ABB RobotStudio station: welding.rspag

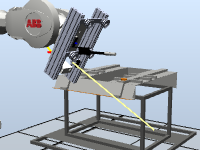
--- station ---
Station Solution21 (saved by RobotStudio format 3)
Controller IRB_7600_340kg_2.80m
  mechanical unit ROB_1: IRB7600_340_280__01, 6 joints, base frame (0, 0, 0) mm
Layout (positions relative to the parent item):
  - IRB7600_340_280__01 [mechanism, from Robots\IRB7600_340_280_G_01.rslib] at (0, 0, 0) mm; joint values [0, 0, 0, 0, 0.5236, 0] (rad or m)
  - Car Underbody [part]
  - Welding Gun [graphiccomponentgroup, from Libraries\Welding Gun.rslib] at (1932.51, 0, 1895) mm, rotated rx 180 ry 60 rz 180 deg
    - Part_1 [part, from Libraries\Welding Gun.rslib]
    - Part_2 [part, from Libraries\Welding Gun.rslib] at (-42.64, -13.71, 48.01) mm
    - Part_3 [part, from Libraries\Welding Gun.rslib] at (-42.16, -13.66, 198.7) mm, rotated rx 0 ry 60 rz 0 deg
    - Part_4 [part, from Libraries\Welding Gun.rslib] at (40.8, 0, 127.95) mm, rotated rx 0 ry -30 rz 0 deg
    - Part_6 [part, from Libraries\Welding Gun.rslib] at (-34.66, -7.16, 195.53) mm, rotated rx 0 ry 60 rz 0 deg
    - Part_8 [part, from Libraries\Welding Gun.rslib] at (-8.62, 0, 212.77) mm, rotated rx 0 ry -30 rz 0 deg
    - Part_9 [part, from Libraries\Welding Gun.rslib] at (-87.9, 0, 349.25) mm, rotated rx 0 ry -30 rz 0 deg
    - Part_10 [part, from Libraries\Welding Gun.rslib] at (-111.22, 0, 389.49) mm, rotated rx 0 ry -30 rz 0 deg
    - Part_11 [part, from Libraries\Welding Gun.rslib] at (-118.48, 0, 400.42) mm, rotated rx 0 ry -30 rz 0 deg
  - SC_Lsensor [smart component]
      signals: DI DI_activeLsensor, AO AO_sensedpoint, DO DO_sensorout
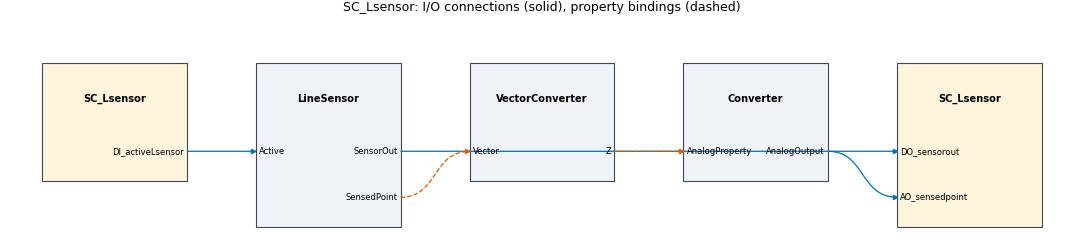
      connections:
        SC_Lsensor.DI_activeLsensor -> LineSensor.Active
        LineSensor.SensorOut -> SC_Lsensor.DO_sensorout
        Converter.AnalogOutput -> SC_Lsensor.AO_sensedpoint
        LineSensor.SensedPoint => VectorConverter.Vector
        VectorConverter.Z => Converter.AnalogProperty
    - VacuumGripper new 12 1 16 [part, from Libraries\VacuumGripper new 12 1 16.rslib] at (1932.51, 0, 1895) mm, rotated rx 0 ry 60 rz 180 deg
    - LineSensor [smart component, from Components\LineSensor.rslib] at (1852.51, 0, 1756.44) mm, rotated rx 180 ry 60 rz 180 deg
        properties: Start=[0 0 0.11]; End=[0 0 1]; Radius=0.001; SensedPart=(none); SensedPoint=[0 0 0]
      - _sensorPart_ [part]
    - Converter [smart component, from Components\Converter.rslib]
        properties: AnalogProperty=0; DigitalProperty=0; BooleanProperty=false; GroupProperty=0
    - VectorConverter [smart component, from Components\VectorConverter.rslib]
        properties: X=0; Y=0; Z=0; Vector=[0 0 0]
Attachment: Part_2 is attached to Part_1
Attachment: Part_3 is attached to Part_1
Attachment: Part_4 is attached to Part_1
Attachment: Part_6 is attached to Part_1
Attachment: Part_8 is attached to Part_1
Attachment: Part_9 is attached to Part_1
Attachment: Part_10 is attached to Part_1
Attachment: Part_11 is attached to Part_1
Attachment: Welding Gun is attached to IRB7600_340_280__01 / Link7
Attachment: VacuumGripper new 12 1 16 is attached to IRB7600_340_280__01 / Link7
Attachment: LineSensor is attached to VacuumGripper new 12 1 16
Station logic (signal -> signal, property => property):
  IRB_7600_340kg_2.80m.ActiveLsensor -> SC_Lsensor.DI_activeLsensor
  SC_Lsensor.AO_sensedpoint -> IRB_7600_340kg_2.80m.AI_sensedpoint
  SC_Lsensor.DO_sensorout -> IRB_7600_340kg_2.80m.DI_sensorOut

--- Backups/IRB_7600_340kg_2.80m/RAPID/TASK1/PROGMOD/CalibData.mod ---
MODULE CalibData
	TASK PERS tooldata welding_gun:=[TRUE,[[0,0,0],[1,0,0,0]],[1,[0,0,1],[1,0,0,0],0,0,0]];
ENDMODULE

--- Backups/IRB_7600_340kg_2.80m/RAPID/TASK1/PROGMOD/Module1.mod ---
MODULE Module1
	CONST robtarget align_tool:=[[1716.000078479,0,1770],[0.000000157,0,1,0],[0,0,0,0],[9E9,9E9,9E9,9E9,9E9,9E9]];
	CONST robtarget Scanfront_edge:=[[35.472465948,1412.646459793,1555.718194742],[0.00647884,0.725347043,-0.688328055,0.005846406],[0,1,1,1],[9E9,9E9,9E9,9E9,9E9,9E9]];

    VAR robtarget next_target;
    VAR robtarget LeftEdgeWithOffsetPlus10;
    VAR robtarget WeldingStartPoint;
    VAR num LeftEdgeWithOffset;
    VAR num LeftEdgeDistance;
    VAR num FrontEdgeWithOffset;
    VAR num FrontEdgeDistance;
    VAR robtarget LeftEdge;
    VAR robtarget FrontEdge;
    CONST speeddata fast_speed:= v1000;
    CONST speeddata slow_speed:= v150;
    CONST speeddata welding_speed:= v30;

    PROC Path_10()
         WaitRob\InPos;
    ENDPROC

    PROC findfront_edge1()
	   MoveJ ScanFront_Edge,fast_speed,fine,tool0\WObj:=wobj0;
        next_target:=Offs(ScanFront_Edge,0,10,0);
         SetDO ActiveLSensor,1;
       WaitRob\InPos;
       WaitTime 0.5;
       FrontEdgeWithOffset:=ai_SensedPoint;
       FrontEdgeDistance:=FrontEdgeWithOffset*1000-ScanFront_Edge.trans.y;

       WHILE TRUE DO
         IF di_SensorOut=0 THEN
            next_target:=Offs(next_target,0,100,0);
             MoveL next_target,fast_speed,fine,tool0\WObj:=wobj0;
            WaitRob\InPos;
       WaitTime 0.5;
         ELSE
             RETURN;
         ENDIF
         ENDWHILE
	ENDPROC

    PROC findfront_edge2()
	WHILE TRUE DO
        IF di_SensorOut=1 THEN
            next_target:=Offs(next_target,0,-50,0);
            MoveL next_target,slow_speed,fine,tool0\WObj:=wobj0;
            WaitRob\InPos;
            WaitTime .1;
        ELSE
            FrontEdge:=next_target;
            RETURN;
        ENDIF
    ENDWHILE
    ENDPROC


    PROC findfront_edge3()
	WHILE TRUE DO
        IF di_SensorOut=0 THEN
            next_target:=Offs(next_target,0,10,0);
            MoveL next_target,slow_speed,fine,tool0\WObj:=wobj0;
            WaitRob\InPos;
            WaitTime .1;
        ELSE
            FrontEdge:=next_target;
            RETURN;
        ENDIF
    ENDWHILE
    ENDPROC





     PROC findfront_edge4()
	WHILE TRUE DO
        IF di_SensorOut=0 THEN
            next_target:=Offs(next_target,0,-0.1,0);
            MoveL next_target,slow_speed,fine,tool0\WObj:=wobj0;
            WaitRob\InPos;
            WaitTime .1;
        ELSE
            FrontEdge:=next_target;
            RETURN;
        ENDIF
    ENDWHILE
    ENDPROC


    PROC findleft_edge1()
	   next_target:=Offs(FrontEdge,0,20,0);
	   MoveL next_target,fast_speed,fine,tool0\WObj:=wobj0;

       SetDO ActiveLSensor,1;
       WaitRob\InPos;
       WaitTime 0.5;
       LeftEdgeWithOffset:=ai_SensedPoint;
       LeftEdgeDistance:=LeftEdgeWithOffset*1000- next_target.trans.x;

     WHILE TRUE DO
         IF di_SensorOut=1 THEN
            next_target:=Offs(next_target,-100,0,0);
            MoveL next_target,fast_speed,fine,tool0\WObj:=wobj0;
            WaitRob\InPos;
        WaitTime 0.5;
         ELSE
             RETURN;
         ENDIF
         ENDWHILE

	ENDPROC

     PROC findleft_edge2()
	WHILE TRUE DO
        IF di_SensorOut=0 THEN
            next_target:=Offs(next_target,50,0,0);
            MoveL next_target,slow_speed,fine,tool0\WObj:=wobj0;
            WaitRob\InPos;
            WaitTime .1;
        ELSE
            LeftEdge:=next_target;
            RETURN;
        ENDIF
    ENDWHILE
    ENDPROC

    PROC findleft_edge3()
	WHILE TRUE DO
        IF di_SensorOut=1 THEN
            next_target:=Offs(next_target,-10,0,0);
            MoveL next_target,slow_speed,fine,tool0\WObj:=wobj0;
            WaitRob\InPos;
            WaitTime .1;
        ELSE
            LeftEdge:=next_target;
            RETURN;
        ENDIF
    ENDWHILE
    ENDPROC

    PROC findleft_edge4()
	WHILE TRUE DO
        IF di_SensorOut=1 THEN
            next_target:=Offs(next_target,-0.1,0,0);
            MoveL next_target,slow_speed,fine,tool0\WObj:=wobj0;
            WaitRob\InPos;
            WaitTime .1;
        ELSE
            LeftEdge:=next_target;
            RETURN;
        ENDIF
    ENDWHILE
    ENDPROC

     PROC Welding()
        SetDO ActiveLSensor,0;
        MoveJ ScanFront_Edge,fast_speed,fine,tool0\WObj:=wobj0;
        LeftEdgeWithOffsetPlus10:=Offs(LeftEdge,10,0,0);
       MoveL RelTool (LeftEdgeWithOffsetPlus10,300,10,190),slow_speed, fine, welding_gun;
       WaitTime 1;
       next_target:=WeldingStartPoint;
       WeldingStartPoint := CRobT(\Tool:=welding_gun \WObj:=wobj0);
       MoveL Offs(WeldingStartPoint,161,0,0),welding_speed,fine,welding_gun\WObj:=wobj0;
       MoveL Offs(WeldingStartPoint,161,0,50),welding_speed,fine,welding_gun\WObj:=wobj0;
       MoveL Offs(WeldingStartPoint,304,0,50),welding_speed,fine,welding_gun\WObj:=wobj0;
       MoveL Offs(WeldingStartPoint,304,0,0),welding_speed,fine,welding_gun\WObj:=wobj0;
       MoveL Offs(WeldingStartPoint,1126,0,0),welding_speed,fine,welding_gun\WObj:=wobj0;
       MoveL Offs(WeldingStartPoint,1126,0,50),welding_speed,fine,welding_gun\WObj:=wobj0;
       MoveL Offs(WeldingStartPoint,1266,0,50),welding_speed,fine,welding_gun\WObj:=wobj0;
       MoveL Offs(WeldingStartPoint,1266,0,0),welding_speed,fine,welding_gun\WObj:=wobj0;
       MoveL Offs(WeldingStartPoint,1430,0,0),welding_speed,fine,welding_gun\WObj:=wobj0;
       MoveJ align_tool,fast_speed,fine,tool0\WObj:=wobj0;
	ENDPROC
    PROC initiate()
        setdo ActiveLSensor,0;

    endproc

    PROC main()
        initiate;
         PATH_10;
         findfront_edge1;
         findfront_edge2;
         findfront_edge3;
         findfront_edge4;
         findleft_edge1;
         findleft_edge2;
         findleft_edge3;
         findleft_edge4;
         Welding;
    ENDPROC

ENDMODULE

--- Backups/IRB_7600_340kg_2.80m/RAPID/TASK1/SYSMOD/LINKEDM.sys ---
%%%
  VERSION:1
  LANGUAGE:ENGLISH
%%%

MODULE LINKEDM (SYSMODULE)

! FOLLOWER
!     Name of electronically linked follower axis used by operator at teach pendent.
      PERS string l_f_axis_name{5}       :=  ["",  "", "", "", ""];

!     Name of the mechanical unit for follower axis.
      PERS string l_f_mecunt_n{5}  :=  ["", "", "", "", ""];

!     Linked follower axis number in the mechanical unit (first axis in mech. unit is number 1).
      PERS num l_f_axis_no{5}      :=  [0,          0,   0,  0,  0];

! MASTER
!     Name of the mechanical unit for linked master axis.
      PERS string l_m_mecunt_n{5} :=  ["", "", "", "", ""];

!     Linked master axis number in the mechanical unit (first axis in mech. unit is number 1).
!     See axis number table in documentation for different master mechanical units.
      PERS num l_m_axis_no{5}     :=  [0,  0,  0,  0,  0];

! POSITION OFFSET
!     The increase of the allowed offset position between the master and follower
!     positions, used when starting AUTO mode. As soon as the offset is decreased
!     the old configurated parameter is used.
!     Example: 3 => the configurated value of allowed offset is increased 3 times.
      PERS num offset_ratio{5}       :=  [10,  10,   10,  10,  10];

! SPEED RATIO
!     Speed_ratio used in AUTO and JOG modes [ very_slow   slow    normal    fast]
!     Value 1 = max allowed manual speed.
      CONST num speed_ratio {20}      := [0.01, 0.01, 0.01, 0.01, 0.01,
                                          0.05, 0.05, 0.05, 0.05, 0.05,
                                          0.20, 0.20, 0.20, 0.20, 0.20,
                                          1.00, 1.00, 1.00, 1.00, 1.00];

! STEP SIZE
!     Displacement position used in JOG mode for each activation of positive or
!     negative movement.                  [very_short    short   normal   long]
!     Unit degees or meter.
      CONST num displacement {20}     := [0.001, 0.001, 0.001, 0.001, 0.001,
                                          0.005, 0.005, 0.005, 0.005, 0.005,
                                          0.020, 0.020, 0.020, 0.020, 0.020,
                                          0.100, 0.100, 0.100, 0.100, 0.100];


!-------------------------------------------------------------
 PROC Linked_m ()
      Linked_m_exe ;
 ENDPROC
ENDMODULE

--- Backups/IRB_7600_340kg_2.80m/SYSPAR/EIO.cfg ---
EIO:CFG_1.0:6:1::
#
EIO_SIGNAL:

      -Name "ActiveLsensor" -SignalType "DO" -Access "All"

      -Name "AI_sensedpoint" -SignalType "AI" -Access "All"

      -Name "DI_sensorOut" -SignalType "DI" -Access "All"
